INTERFACE I_RpcDynamicConfigAmsPort

METHOD WithAmsPort : I_RpcDynamicConfigSymbolPath
VAR_INPUT
	nAmsPort	: T_AmsPort;
END_VAR
END_METHOD

END_INTERFACE

(* stored: Version 1.1.0.1, ProductVersion 3.1.4024.12
   Itf I_RpcDynamicConfigAmsPort: Id {75145a11-3559-438b-aa54-2b1ad70c400b}
   Method WithAmsPort: Id {c0d46c0a-576a-4726-9736-677358b08960} *)
